(* PLC project double_acting_jack, Dassault Systèmes ControlBuild 2024x *)
(* stored: creationDateTime 2023-10-03T11:13:07-01:00 *)

(* This module simulates a double-acting jack driven by a five-way, two positions control valve *)
FUNCTION_BLOCK equipment_library.double_acting_jack
  VAR_INPUT
    energy : BOOL := true;
    cmdSupply : BOOL := true;
    sensorSupply : BOOL := true;
  END_VAR
  VAR_INPUT
    valveWork : BOOL := false;
    valveRest : BOOL := false;
  END_VAR
  VAR_OUTPUT
    outletSensor : BOOL := false;
    inletSensor : BOOL := false;
  END_VAR
  VAR_OUTPUT
    rodPosition : REAL := 0.0;
    rodPercent : REAL := 0.0;
    incrementValue : REAL := 0.0;
  END_VAR
  VAR
    slidePosition : DINT := 0;
    pipeWork : BOOL := false;
    pipeRest : BOOL := true;
    increment : REAL := 0.0;
  END_VAR
  VAR CONSTANT
    outletSensorLogic : BOOL := true;
    inletSensorLogic : BOOL := true;
    rodLength : REAL := 1000.0;
    time2extend : REAL := 2.0;
  END_VAR
  VAR
    d_locking : BOOL := false;
    v_d_locking : REAL := 2.0;
    d_inletSensor : BOOL := false;
    v_d_inletSensor : BOOL := false;
    d_outletSensor : BOOL := false;
    v_d_outletSensor : BOOL := false;
  END_VAR


ACTION C_source_code:
/* ----------------------------------------------------------------	*/
/* Type : Model of Operative Behaviour					*/
/* Category :  Associations - Jacks					*/
/* Author : Dassault Systemes						*/
/* Update date : June 2018							*/
/* ----------------------------------------------------------------	*/
/* This module simulates a double-acting jack driven by a   		*/
/* five-way, two positions control valve .				*/
/* ----------------------------------------------------------------	*/

/* ----------------------------------------------------------------	*/
/* Management of orders from Control Part					*/
/*	if there is no power supply for command the solenoid 		*/
/*     control valve doesn't understand the control order.		*/
/* Hypothesis : if the two control valves are excited at the 		*/
/* same time, only the first is taken into account.			*/
/* ----------------------------------------------------------------	*/
if (cmdSupply && valveWork && ! valveRest) slidePosition=1;
if (cmdSupply &&  ! valveWork && valveRest) slidePosition=0;

/* ----------------------------------------------------------------	*/
/* Calculation of the on-state of the energy in the pipes		*/
/*     if there is no energy in input, pipes are not 			*/
/*	   under pressure.							*/
/* ----------------------------------------------------------------	*/
pipeWork = (slidePosition==1) & energy;
pipeRest = (slidePosition==0) & energy;

/* ----------------------------------------------------------------	*/
/* Management of the rod evolution						*/
/* the rod stays in its current position if there is no pressure 	*/
/* in the two chambers. 							*/
/* ----------------------------------------------------------------	*/
incrementValue = 0;
if (! d_locking)  {
	if (time2extend > 0.0)
		increment = (rodLength/time2extend)*(CLOCK_PERIOD/1000000);
	if (pipeWork && ! pipeRest) {
		if ( rodPosition < rodLength ) {
			(rodPosition) += increment;
			incrementValue = increment;
		}
		if ( rodPosition > rodLength ) {
			incrementValue -= rodPosition - rodLength;
			rodPosition = rodLength;
		}
	}
	if (pipeRest && ! pipeWork) {
		if ( rodPosition > 0 ) {
			(rodPosition) -= increment;
			incrementValue = increment * -1.0;
		}
		if ( rodPosition < 0.0 ) {
			incrementValue -= rodPosition;
			rodPosition = 0.0;
		}
	}
}

/* ----------------------------------------------------------------	*/
/* Calculation of the rod position in percentage			*/
/* ----------------------------------------------------------------	*/
if (rodLength != 0.0)
	rodPercent = ((rodPosition/rodLength)*100);

/* ----------------------------------------------------------------	*/
/* Management of the sensors state						*/
/* ----------------------------------------------------------------	*/
if (d_outletSensor) outletSensor = v_d_outletSensor;
else
	outletSensor = ((rodPosition >= rodLength) ^ ! outletSensorLogic) && sensorSupply;


if (d_inletSensor) inletSensor = v_d_inletSensor;
else
	inletSensor = ((rodPosition <= 0) ^ ! inletSensorLogic) && sensorSupply;
END_ACTION
END_FUNCTION_BLOCK
